KUKA KRL program: connect3ZeroGravity.src, connect3ZeroGravity.dat

--- connect3ZeroGravity.src ---
&ACCESS RVP
&REL 1
DEF  connect3ZeroGravity( )

DECL INT row, col, targetColumn, targetRow, winningPlayer, currentPlayer, stoneNumber, moveToMake, myInt
DECL INT robotColumn, robotRow
DECL BOOL play
DECL INT board[4,6], playerMoves[6]

;FOLD INI;%{PE}
  ;FOLD BASISTECH INI
    GLOBAL INTERRUPT DECL 3 WHEN $STOPMESS==TRUE DO IR_STOPM ( )
    INTERRUPT ON 3
    BAS (#INITMOV,0 )
  ;ENDFOLD (BASISTECH INI)
  ;FOLD USER INI
    ;Make your modifications here

  ;ENDFOLD (USER INI)
;ENDFOLD (INI)
GRPg_SetStateAndCheck(1,1,0.2,0)
;FOLD PTP HOME  Vel= 100 % DEFAULT;%{PE}%MKUKATPBASIS,%CMOVE,%VPTP,%P 1:PTP, 2:HOME, 3:, 5:100, 7:DEFAULT
$BWDSTART = FALSE
PDAT_ACT=PDEFAULT
FDAT_ACT=FHOME
BAS (#PTP_PARAMS,100 )
$H_POS=XHOME
PTP  XHOME
;ENDFOLD
; initialize global values

dX = 47
dY = 32
dZ = 120
play = TRUE

FOR myInt=1 TO 6 STEP 1
   playerMoves[myInt]=-1
ENDFOR



; ---------- PREPARE BOARD WITH STONES -------

; prepareBoard()


; --------------------------------------------
; ---------- 3 START OF THE PROGRAM ----------

; Restart Start -------------
WHILE play == TRUE

   ; ----------  FILL BOARD WITH ZEROS ----------
   row = 1
   col = 1
   FOR row=1 TO boardRows STEP 1
      FOR col=1 TO boardColumns STEP 1
         board[row, col]=0
      ENDFOR
   ENDFOR

   stoneNumber = 1
   currentPlayer = -1
   moveToMake = -1
   targetColumn = -1
   targetRow = -1

   startingPlayer = player_question()
   ; 1 = Human starts, 2 = Robot starts

   IF (startingPlayer == 1) THEN
       WHILE (checkWinner(board[,]) == -1)
           targetColumn = col_question()
           targetRow = row_question()
          ; Place block for player
           board[targetRow, targetColumn] = 1
           placeStone(targetRow, targetColumn, 1, stoneNumber)
           IF (checkWinner(board[,]) <> -1) THEN
               EXIT
           ENDIF
           ; calculate robot response
           ; !!!TARGETROW IS WRONG!!!
           robotColumn = calculateRobotResponse(board[,], targetColumn)
           robotRow = checkRow(board[,], robotColumn)
           board[robotRow, robotColumn] = 2
           placeStone(robotRow, robotColumn, 2, stoneNumber)
           stoneNumber = stoneNumber + 1
       ENDWHILE
   ENDIF

   IF (startingPlayer == 2) THEN
      targetColumn = 4
      WHILE (checkWinner(board[,]) == -1)
        ; calculate robot response
        ; !!!TARGETROW IS WRONG!!!
        robotColumn = calculateRobotResponse(board[,], targetColumn)
        robotRow = checkRow(board[,], robotColumn)
        board[robotRow, robotColumn] = 2
        placeStone(robotRow, robotColumn, 2, stoneNumber)
        IF (checkWinner(board[,]) <> -1) THEN
            EXIT
        ENDIF
         ; Get humans move
        targetColumn = col_question()
        targetRow = row_question()
        ; Place block for player
        board[targetRow, targetColumn] = 1
        placeStone(targetRow, targetColumn, 1, stoneNumber)
        stoneNumber = stoneNumber + 1
      ENDWHILE
   ENDIF

;   IF (startingPlayer == 2) THEN
;      WHILE (checkWinner(board[,]) == -1)
;
;         ; Calulate robots move
;         moveToMake = getOptimalMove(targetColumn, stoneNumber, playerMoves[1], playerMoves[3])
;
;         targetRow = checkRow(board[,], moveToMake)
;         board[targetRow, moveToMake] = 2
;         placeStone(targetRow, moveToMake, 2, stoneNumber)
;        IF (checkWinner(board[,]) <> -1) THEN
;            EXIT
;        ENDIF
;         ; Get humans move
;         targetColumn = col_question()
;         targetRow = checkRow(board[,], targetColumn)
;         board[targetRow, targetColumn] = 1
;         placeStone(targetRow, targetColumn, 1, stoneNumber)
;         playerMoves[stoneNumber] = targetColumn
;         stoneNumber = stoneNumber + 1
;      ENDWHILE
;   ENDIF

   ; Print the winner is Player
   winningPlayer = checkWinner(board[,])
   winnerAnnouncement(winningPlayer)

   ; Do you want to play again?

   IF playAgainQuestion() == 1 THEN
      play = TRUE
   ELSE
      play = FALSE
   ENDIF
   cleanUp(board[,])

ENDWHILE




;FOLD PTP HOME  Vel= 100 % DEFAULT;%{PE}%MKUKATPBASIS,%CMOVE,%VPTP,%P 1:PTP, 2:HOME, 3:, 5:100, 7:DEFAULT
$BWDSTART = FALSE
PDAT_ACT=PDEFAULT
FDAT_ACT=FHOME
BAS (#PTP_PARAMS,100 )
$H_POS=XHOME
PTP  XHOME
;ENDFOLD

END

DEF placeStone(row1:IN, targetColumn1:IN, currentPlayer1:IN, stoneNumber1:IN)
   DECL INT targetColumn1, currentPlayer1, stoneNumber1, row1
   DECL FRAME placePosition, upPosition

   pickstoneFromBoard (currentPlayer1, stoneNumber1)

   placePosition = XP1
   placePosition.X = placePosition.X + (targetColumn1-1)*dX
   placePosition.Y = placePosition.Y + (row1-1)*dY
   upPosition = placePosition
   upPosition.Z = upPosition.Z + dZ
   $TOOL = TOOL_DATA[14]
   $BASE = BASE_DATA[5]
   SPTP upPosition
   SLIN placePosition
   GRPg_SetStateAndCheck(1,1,0.2,0)
   SLIN upPosition
END

--- connect3ZeroGravity.dat ---
&ACCESS RVP
&REL 1
DEFDAT  connect3ZeroGravity
;FOLD EXTERNAL DECLARATIONS;%{PE}%MKUKATPBASIS,%CEXT,%VCOMMON,%P
;FOLD BASISTECH EXT;%{PE}%MKUKATPBASIS,%CEXT,%VEXT,%P
EXT  BAS (BAS_COMMAND  :IN,REAL  :IN )
DECL INT SUCCESS
;ENDFOLD (BASISTECH EXT)
;FOLD USER EXT;%{E}%MKUKATPUSER,%CEXT,%VEXT,%P
;Make your modifications here

DECL INT column,player,startingPlayer
DECL REAL dX,dY,dZ
;ENDFOLD (USER EXT)
;ENDFOLD (EXTERNAL DECLARATIONS)
DECL E6POS XP1={X -113.396988,Y 57.0544930,Z -34.5422562,A -105.776718,B 88.3243942,C -17.1389370,S 2,T 10,E1 0.0,E2 0.0,E3 0.0,E4 0.0,E5 0.0,E6 0.0}
DECL FDAT FP1={TOOL_NO 14,BASE_NO 5,IPO_FRAME #BASE,POINT2[] " ",TQ_STATE FALSE}
ENDDAT
